PROGRAM MAIN
VAR
	mqtt: MQTT;
	
	tonTimer : TON := (PT:=T#10S); //Interval timer for broadcasting.
	ton1sTimer : TON := (PT:=T#1S);
END_VAR

IF _TaskInfo[GETCURTASKINDEXEX()].FirstCycle THEN
	mqtt.configureMQTTClient();
END_IF 
mqtt.connect();
 
mqtt.publishWithTON(timer:=tonTimer, msg:='hi there!');
mqtt.publishWithTON(timer:=ton1sTimer, msg:='1s');

END_PROGRAM

(* stored: Version 1.1.0.1, ProductVersion 3.1.4024.11
   POU MAIN: Id {bcad94f3-26d4-4398-99c6-2ab4d243b808}, SpecialFunc None *)
